TYPE ST_PiezoStagePP EXTENDS ST_PiezoStage :
STRUCT
    (* Global variables for the RPDO data to the drive. Each one is linked to the respective RPDO channel. *)
    nProfilVelocity 		AT %Q* : DINT;
    nProfilAcceleration		AT %Q* : DINT;
    nProfilDecceleration	AT %Q* : DINT;

END_STRUCT
END_TYPE

(* stored: Version 1.1.0.1
   DUT ST_PiezoStagePP: Id {f3138ec3-c7d2-4909-8437-b2c9f6ce683d} *)
